// TIA Portal V15 export
// export: Created 2018-05-29T12:25:38.1552518Z, ExportSetting WithDefaults, DisplayName Totally Integrated Automation Portal, DisplayVersion V15, DisplayName STEP 7 Professional, DisplayVersion V15, DisplayName WinCC Professional, DisplayVersion V15, DisplayName TIA Portal Openness, DisplayVersion V15
FUNCTION "XV501_fc" : Void   // FC1, STL
TITLE = XV501_fc
{ S7_Optimized_Access := 'TRUE' }
VERSION : 0.1
// Some Valve  on drawing 20 test
// stored: AutoNumber true, UDAEnableTagReadback false
BEGIN

NETWORK
TITLE = Main
// comment: PLC1


// Call the CM FB with the corresponding DB instance
      CALL  "BST_VALVE_400", "XV501"
      ( AUT_OP   := ,
        FB_OPEN  := ,
        FB_CLOSE := ,
        QOPEN    := ,
        QCLOSE   := ,
        QMON_ERR := ,
        QCMD_OP  := 
      );
END_FUNCTION
